TYPE String_Array256 :
UNION
	sValue			:STRING; 
	arrByte 		:ARRAY[0..255] OF BYTE;
END_UNION
END_TYPE

(* stored: Version 1.1.0.1
   DUT String_Array256: Id {0ee99773-9d8c-49a1-95a8-e80c42c3007b} *)
